PROGRAM POU
VAR
END_VAR

END_PROGRAM

(* stored: Version 1.1.0.1, ProductVersion 3.1.4026.18
   POU POU: Id {6a1996b1-e545-449d-bb5b-c30ca6a6df6e}, SpecialFunc None *)
